ABB RobotStudio station: Proyecto_Final_B2_20210602-202218.rsstn

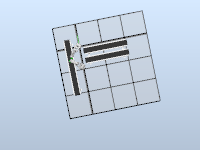
Station Station (saved by RobotStudio 20.4.9280.0)
Controller Controlador5, task T_ROB2: task frame (RAPID world) sits at (0, 0, 300) mm in the station
Controller Controlador5, task T_ROB1: task frame (RAPID world) sits at (0, 0, 300) mm in the station
Controller Controlador5
  mechanical unit ROB_1: IRB120_3_58__01, 6 joints, base frame (0, 0, 0) mm
  mechanical unit ROB_2: IRB120_3_58__01_2, 6 joints, base frame (0, -900, 0) mm
Layout (positions relative to the parent item):
  - IRB120_3_58__01 [mechanism, from Robots\IRB120_3_58_G_01.rslib] at (0, 0, 300) mm; joint values [-2.3296, 1.1697, -0.7465, -0.0449, 0.9342, 0.5131] (rad or m)
  - Belt Conveyor [part]
  - Belt Conveyor [part]
  - IRB120_3_58__01_2 [mechanism, from Robots\IRB120_3_58_G_01.rslib] at (0, -900, 300) mm; joint values [2.464, 1.1375, -0.7171, 0.028, 0.9016, 0] (rad or m)
  - Belt Conveyor [part]
